// TIA Portal V20 export
TYPE "StationLight"
   STRUCT
      SensorA : Bool;
      SensorB : Bool;
      SensorC : Bool;
      SensorD : Bool;
      IsEmpty : Bool;
      IsOccupied : Bool;
      Numer : SInt;
   END_STRUCT;
END_TYPE
